PROGRAM PRG_TEST
VAR
    MovingAverage_Test : FB_MovingAverage_Test;
END_VAR

TcUnit.RUN();

END_PROGRAM

(* stored: Version 1.1.0.1, ProductVersion 3.1.4022.16
   POU PRG_TEST: Id {2b0f2396-05a8-4641-ad59-d0377b4454be}, SpecialFunc None *)
